{attribute 'GeneratedUsingTerminal: EJ4002-0000-0017'}
{attribute addProperty BoxType "EJ4002-0000-0017"}
{attribute addProperty Id "Analog_outputAT %Q*INT2"}
{attribute addProperty CRC "3128867708"}
{attribute addProperty Size "2"}
TYPE AO_Outputs_Channel_BA7EBB7C :
STRUCT
	{attribute addProperty Name "Analog_output"}
	Analog_output AT %Q* : INT;
END_STRUCT
END_TYPE

(* stored: Version 1.2.0.0, ProductVersion 3.1.4024.9
   DUT AO_Outputs_Channel_BA7EBB7C: Id {de716554-6e8d-45c3-901d-7e85617809e8} *)
